// TIA Portal project "ProjetoISA5.1" (V19)

(* hardware
DEVICE "S7-1200 station_1"  S7-1200 Station
   slot 0: "Rack_0"  S7-1200 Rack  Rack  V1.0
   slot 1: "PLC_1"  CPU 1215C DC/DC/DC  6ES7 215-1AG40-0XB0  V4.6
*)

// ===== PLC "PLC_1"  CPU 1215C DC/DC/DC =====

VAR_GLOBAL   // PLC tag table "Default tag table"
   "System_Byte" AT %MB1 : Byte;
   "FirstScan" AT %M1.0 : Bool;
   "DiagStatusUpdate" AT %M1.1 : Bool;
   "AlwaysTRUE" AT %M1.2 : Bool;
   "AlwaysFALSE" AT %M1.3 : Bool;
   "Clock_Byte" AT %MB0 : Byte;
   "Clock_10Hz" AT %M0.0 : Bool;
   "Clock_5Hz" AT %M0.1 : Bool;
   "Clock_2.5Hz" AT %M0.2 : Bool;
   "Clock_2Hz" AT %M0.3 : Bool;
   "Clock_1.25Hz" AT %M0.4 : Bool;
   "Clock_1Hz" AT %M0.5 : Bool;
   "Clock_0.625Hz" AT %M0.6 : Bool;
   "Clock_0.5Hz" AT %M0.7 : Bool;
END_VAR

VAR_GLOBAL   // PLC tag table "03 - EntradasAnalógicas"
   "MIW_FT01" AT %IW64 : Int;   // Transmissor de Vazão
   "MIW_LT01" AT %IW66 : Int;
END_VAR

VAR_GLOBAL   // PLC tag table "02 - SaidasDigitais"
   "MQ_LigaInversor01" AT %Q0.0 : Bool;
END_VAR

VAR_GLOBAL   // PLC tag table "01 - EntradasDigitais"
   "MI_BotEmergencia" AT %I0.0 : Bool;   // Botão de Emergência
   "MI_LSH.TQ01" AT %I0.1 : Bool;   // Nivel Alto Tanque 01
   "MI_LSL.TQ02" AT %I0.2 : Bool;   // Nivel Baixo Tanque 02
   "MI_StatusInversor01" AT %I0.3 : Bool;   // Feedback Inversor 01
END_VAR

DATA_BLOCK "DB01_Espelhamento"   // DB1
{ S7_Optimized_Access := 'FALSE' }
VERSION : 0.1
   VAR
      EntradasDigitais : Struct
         MX_BotEmergencia : Bool;
         MX_LSHTQ1 : Bool;
         MX_LSLTQ2 : Bool;
         MX_StatusInversor01 : Bool;
      END_STRUCT;
      SaidasDigitais : Struct
         MX_LigaInversor01 : Bool;
      END_STRUCT;
      EntradasAnalogicas : Struct
         MW_FT01 : DInt;
         MW_LT01 : DInt;
      END_STRUCT;
   END_VAR
BEGIN
END_DATA_BLOCK

DATA_BLOCK "DB02_Operacao"   // DB2
{ S7_Optimized_Access := 'FALSE' }
VERSION : 0.1
   VAR
      MX_StatusOperacao : Bool;
   END_VAR
BEGIN
END_DATA_BLOCK

DATA_BLOCK "FB01_PartidaMotor_DB"   // DB3
{ S7_Optimized_Access := 'TRUE' }
VERSION : 0.1
// stored: InstanceOfName FB01_PartidaMotor
"FB01_PartidaMotor"
BEGIN
END_DATA_BLOCK

DATA_BLOCK "DB03_IHM"   // DB4
{ S7_Optimized_Access := 'FALSE' }
VERSION : 0.1
   VAR
      MX_LigaManualBomba01 : Bool;
      MX_LigaAutomaticoBomba01 : Bool;
   END_VAR
BEGIN
END_DATA_BLOCK

DATA_BLOCK "FB01_PartidaMotor_DB_1"   // DB5
{ S7_Optimized_Access := 'TRUE' }
VERSION : 0.1
// stored: InstanceOfName FB01_PartidaMotor
"FB01_PartidaMotor"
BEGIN
END_DATA_BLOCK

DATA_BLOCK "DB04_ParametrizacaoAnalogica"   // DB6
{ S7_Optimized_Access := 'FALSE' }
VERSION : 0.1
   VAR
      MW_MinFT01 : Real;
      MW_MaxFT01 : Real;
      MW_MinLT01 : Real;
      MW_MaxLT01 : Real;
      MW_ValueFT01 : Real;
      MW_ValueLT01 : Real;
   END_VAR
BEGIN
END_DATA_BLOCK

FUNCTION_BLOCK "FB01_PartidaMotor"   // FB1, LAD
{ S7_Optimized_Access := 'TRUE' }
VERSION : 0.1
   VAR_INPUT
      Emergencia : Bool;
      Automatico : Bool;
      Manual : Bool;
      LSH : Bool;
      LSL : Bool;
   END_VAR
   VAR_OUTPUT
      LigaMotor : Bool;
   END_VAR
BEGIN

REGION Network 1
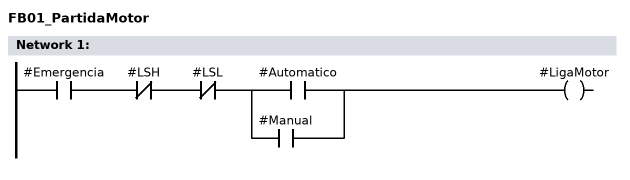
   RUNG wire#powerrail
      Contact( #Emergencia )
      I_Contact( #LSH )
      I_Contact( #LSL )
      wire#w1
      Contact( #Automatico )
      wire#w2
      Coil( #LigaMotor )
   END_RUNG
   RUNG wire#w1
      Contact( #Manual )
   END_RUNG wire#w2
   // the same network as SCL:
   #LigaMotor := #Emergencia AND NOT #LSH AND NOT #LSL AND (#Automatico OR #Manual);
END_REGION
END_FUNCTION_BLOCK

FUNCTION "FC01.0_EntradaDigitais" : Void   // FC1, SCL
{ S7_Optimized_Access := 'TRUE' }
VERSION : 0.1
BEGIN
   REGION Entradas_Digitais_CPU
       "DB01_Espelhamento".EntradasDigitais.MX_BotEmergencia := "MI_BotEmergencia";
       "DB01_Espelhamento".EntradasDigitais.MX_LSHTQ1 := "MI_LSH.TQ01";
       "DB01_Espelhamento".EntradasDigitais.MX_LSLTQ2 := "MI_LSL.TQ02";
       "DB01_Espelhamento".EntradasDigitais.MX_StatusInversor01 := "MI_StatusInversor01";

   END_REGION
END_FUNCTION

FUNCTION "FC01.1_SaidasDigitais" : Void   // FC2, SCL
{ S7_Optimized_Access := 'TRUE' }
VERSION : 0.1
BEGIN
   REGION Saidas_Digitais_CPU
       "MQ_LigaInversor01" := "DB01_Espelhamento".SaidasDigitais.MX_LigaInversor01;

   END_REGION
END_FUNCTION

FUNCTION "FC01.2_EntradasAnalogicas" : Void   // FC3, SCL
{ S7_Optimized_Access := 'TRUE' }
VERSION : 0.1
BEGIN
   REGION Entradas_Analogicas_CPU
       "DB01_Espelhamento".EntradasAnalogicas.MW_FT01 := "MIW_FT01";
       "DB01_Espelhamento".EntradasAnalogicas.MW_LT01 := "MIW_LT01";

   END_REGION
END_FUNCTION

FUNCTION "FC02.0_Emergencia" : Void   // FC4, LAD
{ S7_Optimized_Access := 'TRUE' }
VERSION : 0.1
   VAR_TEMP
      StatusEmergencia : Bool;
   END_VAR
BEGIN

REGION Network 1
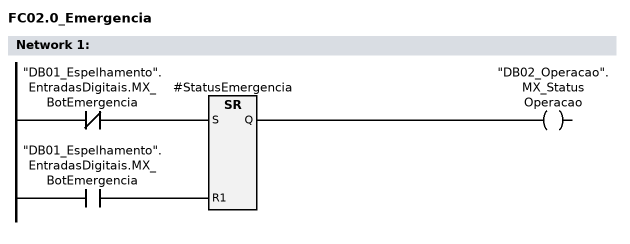
   RUNG wire#powerrail
      I_Contact( "DB01_Espelhamento".EntradasDigitais.MX_BotEmergencia )
      S_SR(operand := #StatusEmergencia, r1 := wire#w1)
      Coil( "DB02_Operacao".MX_StatusOperacao )
   END_RUNG
   RUNG wire#powerrail
      Contact( "DB01_Espelhamento".EntradasDigitais.MX_BotEmergencia )
   END_RUNG wire#w1
   // the same network as SCL:
   IF NOT "DB01_Espelhamento".EntradasDigitais.MX_BotEmergencia THEN
       #StatusEmergencia := TRUE;   // SR flip-flop
   END_IF;
   IF "DB01_Espelhamento".EntradasDigitais.MX_BotEmergencia THEN #StatusEmergencia := FALSE; END_IF;
   "DB02_Operacao".MX_StatusOperacao := #StatusEmergencia;
END_REGION
END_FUNCTION

FUNCTION "FC03_Operacao" : Void   // FC5, LAD
{ S7_Optimized_Access := 'TRUE' }
VERSION : 0.1
BEGIN

REGION Network 1
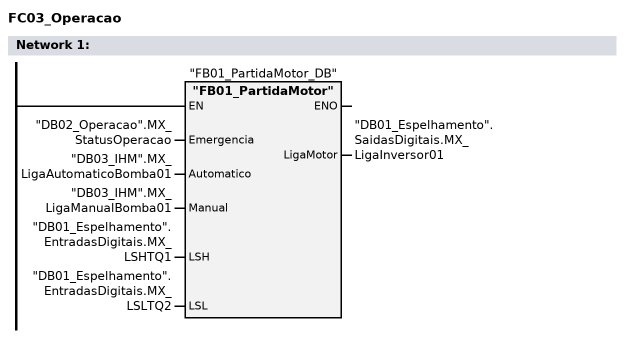
   RUNG wire#powerrail
      "FB01_PartidaMotor_DB"(Emergencia := "DB02_Operacao".MX_StatusOperacao, Automatico := "DB03_IHM".MX_LigaAutomaticoBomba01, Manual := "DB03_IHM".MX_LigaManualBomba01, LSH := "DB01_Espelhamento".EntradasDigitais.MX_LSHTQ1, LSL := "DB01_Espelhamento".EntradasDigitais.MX_LSLTQ2, LigaMotor => "DB01_Espelhamento".SaidasDigitais.MX_LigaInversor01)
   END_RUNG
   // the same network as SCL:
   "FB01_PartidaMotor_DB"(Emergencia := "DB02_Operacao".MX_StatusOperacao,   // "FB01_PartidaMotor"
                          Automatico := "DB03_IHM".MX_LigaAutomaticoBomba01,
                          Manual := "DB03_IHM".MX_LigaManualBomba01,
                          LSH := "DB01_Espelhamento".EntradasDigitais.MX_LSHTQ1,
                          LSL := "DB01_Espelhamento".EntradasDigitais.MX_LSLTQ2,
                          LigaMotor => "DB01_Espelhamento".SaidasDigitais.MX_LigaInversor01);
END_REGION
END_FUNCTION

FUNCTION "FC04_Analogicas" : Void   // FC6, LAD
{ S7_Optimized_Access := 'TRUE' }
VERSION : 0.1
   VAR_TEMP
      FTNormX : Real;
      LTNormX : Real;
   END_VAR
BEGIN

REGION Network 1: Transmissor de Vazão
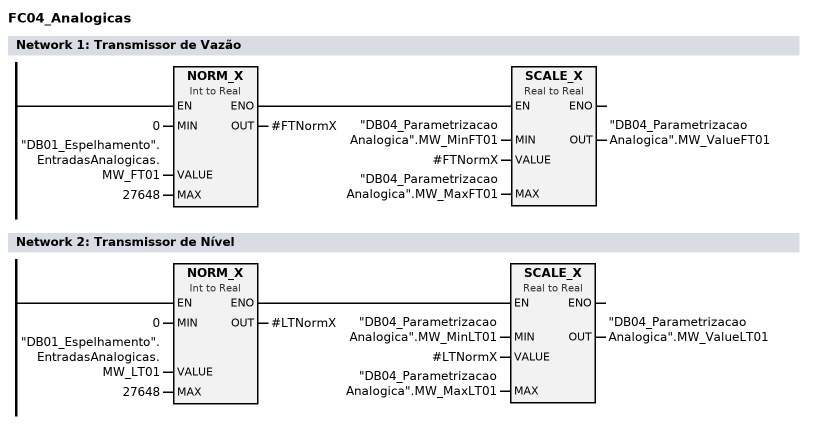
   RUNG wire#powerrail
      { S7_Templates := "[SrcType := Int, DestType := Real]" } Normalize(min := 0, value := "DB01_Espelhamento".EntradasAnalogicas.MW_FT01, max := 27648, out => #FTNormX)
      { S7_Templates := "[SrcType := Real, DestType := Real]" } Scale(min := "DB04_ParametrizacaoAnalogica".MW_MinFT01, value := #FTNormX, max := "DB04_ParametrizacaoAnalogica".MW_MaxFT01, out => "DB04_ParametrizacaoAnalogica".MW_ValueFT01)
   END_RUNG
   // the same network as SCL:
   #FTNormX := NORM_X(MIN := 0, VALUE := "DB01_Espelhamento".EntradasAnalogicas.MW_FT01, MAX := 27648);
   "DB04_ParametrizacaoAnalogica".MW_ValueFT01 := SCALE_X(MIN := "DB04_ParametrizacaoAnalogica".MW_MinFT01, VALUE := #FTNormX, MAX := "DB04_ParametrizacaoAnalogica".MW_MaxFT01);
END_REGION

REGION Network 2: Transmissor de Nível
   RUNG wire#powerrail
      { S7_Templates := "[SrcType := Int, DestType := Real]" } Normalize(min := 0, value := "DB01_Espelhamento".EntradasAnalogicas.MW_LT01, max := 27648, out => #LTNormX)
      { S7_Templates := "[SrcType := Real, DestType := Real]" } Scale(min := "DB04_ParametrizacaoAnalogica".MW_MinLT01, value := #LTNormX, max := "DB04_ParametrizacaoAnalogica".MW_MaxLT01, out => "DB04_ParametrizacaoAnalogica".MW_ValueLT01)
   END_RUNG
   // the same network as SCL:
   #LTNormX := NORM_X(MIN := 0, VALUE := "DB01_Espelhamento".EntradasAnalogicas.MW_LT01, MAX := 27648);
   "DB04_ParametrizacaoAnalogica".MW_ValueLT01 := SCALE_X(MIN := "DB04_ParametrizacaoAnalogica".MW_MinLT01, VALUE := #LTNormX, MAX := "DB04_ParametrizacaoAnalogica".MW_MaxLT01);
END_REGION
END_FUNCTION

ORGANIZATION_BLOCK "Main"   // OB1, LAD, ProgramCycle
TITLE = "Main Program Sweep (Cycle)"
{ S7_Optimized_Access := 'TRUE' }
VERSION : 0.1
   VAR_INPUT
      Initial_Call : Bool;   // Initial call of this OB
      Remanence : Bool;   // =True, if remanent data are available
   END_VAR
BEGIN
END_ORGANIZATION_BLOCK